Staubli VAL3: clkAirexOn.pgx

program clkAirexOn()
  local num idx
begin

  for idx = 0 to 5
    if statusValves[airexValve[idx]] == 0
      call toggleValve(airexValve[idx])
    endIf
  endFor

end
